{attribute 'linkalways'} 
{attribute 'no_explicit_call' := 'This FB is a CLASS and must be accessed using methods or properties'}
{attribute 'enable_dynamic_creation'}
FUNCTION_BLOCK Node_F_VN_AppendToContainer_TcVnDMatch EXTENDS VisionNode
VAR
    stElement : _TcVnDMatch;
    ipContainer : _ITcVnContainer;
    hrPrev : _HRESULT(S_OK);
	hresult : _HRESULT(S_OK);
END_VAR

METHOD PUBLIC  Clone : I_Node
VAR
	pNode : POINTER TO Node_F_VN_AppendToContainer_TcVnDMatch;
END_VAR
pNode := __NEW(Node_F_VN_AppendToContainer_TcVnDMatch);
Clone := pNode^;
END_METHOD

METHOD FB_init : BOOL
VAR_INPUT
	bInitRetains : BOOL; // if TRUE, the retain variables are initialized (warm start / cold start)
	bInCopyCode : BOOL;  // if TRUE, the instance afterwards gets moved into the copy code (online change)
END_VAR
AddInput('stElement', stElement);
AddInput('ipContainer', ipContainer);
AddInput('hrPrev', hrPrev);
AddOutput('ipContainer', ipContainer);
AddOutput('hresult',hresult);
END_METHOD

METHOD PROTECTED OnExecute
hresult.Value := F_VN_AppendToContainer_TcVnDMatch(
    stElement := stElement.Value,
	ipContainer := ipContainer.Value,
	hrPrev:= hrPrev.Value);
END_METHOD

METHOD PUBLIC PreExecutionCheck
VAR_INPUT
	Check : I_PreExecutionChecks;
END_VAR
Check.IsTrue(ipContainer.IsValid, 'ipContainer must be a valid container');
Check.IsTrue(ipContainer.IsType(TC_GLOBAL_CONST_LIST.ContainerType_Vector_TcVnDMatch), 'ipContainer contains incorrect type');
END_METHOD

END_FUNCTION_BLOCK

(* stored: Version 1.1.0.1, ProductVersion 3.1.4026.13
   POU Node_F_VN_AppendToContainer_TcVnDMatch: Id {4c4c7612-5869-0cbd-357d-daa7778ab2a3}, SpecialFunc None
   Folder Constructor: Id {ccbda210-dd27-011d-09cd-53be85873263}
   Method Clone: Id {8896af77-e9ee-07ce-0f10-9556b7122ed0}
   Method FB_init: Id {bf4736e6-3b80-0656-3b4b-7d68f2417f51}
   Method OnExecute: Id {85026f73-291f-054f-2d47-c2431a5e20b3}
   Method PreExecutionCheck: Id {9921916d-a1ff-0992-0648-24dacf99f32b} *)
